// TwinCAT 3 PLC project tc3test
// ProgramVersion: 3.1.4026.21
// libraries:
//   Tc2_Standard, * (Beckhoff Automation GmbH)
//   Tc2_System, * (Beckhoff Automation GmbH)
//   [Tc3_Base], * (Daniel Wiege)
// project tree:
//   0_Core/ FB_Program.TcPOU (not stored), GVL_Program.TcGVL, Prg_FastCall.TcPOU, Prg_MainCall.TcPOU, TaskFast.TcTTO, TaskMain.TcTTO
// real-time tasks:
//   TASK TaskMain: cycle T#10ms, priority 20, ADS port 350
//   TASK TaskFast: cycle T#10ms, priority 1, ADS port 351

CONFIGURATION tc3test
    RESOURCE PLC ON TwinCAT3
        TASK TaskFast(INTERVAL := T#10ms, PRIORITY := 1);
        TASK TaskMain(INTERVAL := T#10ms, PRIORITY := 20);
        PROGRAM Prg_FastCall WITH TaskFast : Prg_FastCall;
        PROGRAM Prg_MainCall WITH TaskMain : Prg_MainCall;
    END_RESOURCE
END_CONFIGURATION

// ---- 0_Core/GVL_Program.TcGVL
VAR_GLOBAL
	Prg				: FB_Program(0);
END_VAR

// ---- 0_Core/Prg_FastCall.TcPOU
PROGRAM Prg_FastCall

Prg.FastCall();

END_PROGRAM

// ---- 0_Core/Prg_MainCall.TcPOU
PROGRAM Prg_MainCall

Prg.MainCall();

END_PROGRAM
